{attribute 'linkalways'} 
{attribute 'no_explicit_call' := 'This FB is a CLASS and must be accessed using methods or properties'}
{attribute 'enable_dynamic_creation'}
FUNCTION_BLOCK _STRING EXTENDS DatatypeBase
VAR
	localData : T_MaxString;
	activeData : REFERENCE TO T_MaxString REF= localData;
END_VAR

PROPERTY PUBLIC Address : PVOID
GET
Address := ADR(activeData);
END_GET
END_PROPERTY

METHOD PUBLIC ClearReference
VAR_INPUT
END_VAR
activeData REF= localData;
END_METHOD

METHOD PUBLIC Clone : I_Datatype
VAR
    pClone : POINTER TO _STRING;
END_VAR
pClone := __NEW(_STRING(InitialValue := Value));
Clone := pClone^;
END_METHOD

METHOD FB_init : BOOL
VAR_INPUT
	bInitRetains : BOOL; // if TRUE, the retain variables are initialized (warm start / cold start)
	bInCopyCode : BOOL;  // if TRUE, the instance afterwards gets moved WORDo the copy code (online change)
	InitialValue : T_MaxString;
END_VAR
localData := InitialValue;
END_METHOD

METHOD PUBLIC MakeReferenceTo
VAR_INPUT
	ReferenceTarget : REFERENCE TO T_MaxString;
END_VAR
activeData REF= ReferenceTarget;
END_METHOD

PROPERTY PUBLIC Name : T_MAXSTRING
GET
Name := 'STRING';
END_GET
END_PROPERTY

METHOD PUBLIC SerializeWith
VAR_INPUT
	Serializer : I_Serializer;
END_VAR
Serializer.AddString(activeData);
END_METHOD

PROPERTY PUBLIC Size : UDINT
GET
Size := SIZEOF(activeData);
END_GET
END_PROPERTY

METHOD TryDeserializeFrom : BOOL
VAR_INPUT
	Deserializer : I_Deserializer;
	Feedback : I_DeserializerFeedback;
END_VAR
TryDeserializeFrom := Deserializer.TryGetString(activeData, Feedback);
END_METHOD

METHOD TryMakeReferenceTo : BOOL
VAR_INPUT
	Target : I_Datatype;
END_VAR
VAR
	pTargetData : POINTER TO T_MaxString;
END_VAR
IF NOT (Target.Name = Name) THEN
	RETURN;
END_IF

pTargetData := Target.Address;
activeData REF= pTargetData^;
TryMakeReferenceTo := TRUE;
END_METHOD

PROPERTY PUBLIC Value : T_MaxString
GET
Value := activeData;
END_GET
SET
activeData := Value;
END_SET
END_PROPERTY

END_FUNCTION_BLOCK

(* stored: Version 1.1.0.1, ProductVersion 3.1.4024.12
   POU _STRING: Id {09cc697e-4bf4-0a46-1f9f-a11a8e0c06ff}, SpecialFunc None
   Folder Constructor: Id {37df4712-b3b8-0912-3c7b-b976db156eb2}
   Property Address: Id {894857bf-6ce7-0eca-29e5-ebe475e08a03}
   Get Get: Id {a263627a-9dd0-0a5c-2a74-a0f0b07223f1}
   Method ClearReference: Id {9e0896e0-e8ff-0a40-15ec-ab3376683a35}
   Method Clone: Id {39c883a0-31d7-053d-25ce-0fb5d5814828}
   Method FB_init: Id {dd958409-ce2b-0075-3321-b4759b0d14a4}
   Method MakeReferenceTo: Id {95e34d4a-9a92-0b8c-37fc-46185d96f409}
   Property Name: Id {1c323148-3802-0e58-0533-0a156a959090}
   Get Get: Id {afd28dc2-9810-0e51-04d9-f738234c8e47}
   Method SerializeWith: Id {6f369039-49e5-0aeb-19d6-0ce197b2d7b2}
   Property Size: Id {217689d9-6d36-0e62-1697-99ab7fdb10f0}
   Get Get: Id {7fce20cd-e1b5-0e7d-0ad2-34a639a664da}
   Method TryDeserializeFrom: Id {ccba85c8-a1ee-0d57-019c-5bb14171e887}
   Method TryMakeReferenceTo: Id {fa4eb6d8-d665-025d-30d3-ab04ed390a6c}
   Property Value: Id {c9e6417f-ae47-04e3-3a2e-6943a0858fa0}
   Get Get: Id {266ae04a-bc9b-0dcb-3ce6-a1882c771d9c}
   Set Set: Id {94828e65-54bb-0532-0cbf-546638410bb8} *)
